{attribute 'linkalways'} 
{attribute 'no_explicit_call' := 'This FB is a CLASS and must be accessed using methods or properties'}
{attribute 'enable_dynamic_creation'}
FUNCTION_BLOCK Node_F_VN_WarpPerspective_Point EXTENDS VisionNode
VAR
	aSrcPoint : _TcVnPoint2_LREAL;
    aDestPoint : _TcVnPoint2_LREAL;
    aTransformationMatrix : _TcVnMatrix3x3_LREAL;
    hrPrev : _HRESULT(S_OK);
	hresult : _HRESULT(S_OK);
END_VAR

METHOD PUBLIC  Clone : I_Node
VAR
	pNode : POINTER TO Node_F_VN_WarpPerspective_Point;
END_VAR
pNode := __NEW(Node_F_VN_WarpPerspective_Point);
Clone := pNode^;
END_METHOD

METHOD FB_init : BOOL
VAR_INPUT
	bInitRetains : BOOL; // if TRUE, the retain variables are initialized (warm start / cold start)
	bInCopyCode : BOOL;  // if TRUE, the instance afterwards gets moved into the copy code (online change)
END_VAR
AddInput('aSrcPoint', aSrcPoint);
AddInput('aTransformationMatrix', aTransformationMatrix);
AddInput('hrPrev', hrPrev);
AddOutput('aDestPoint', aDestPoint);
AddOutput('hresult',hresult);
END_METHOD

METHOD PROTECTED OnExecute
hresult.Value := F_VN_WarpPerspective_Point(
	aSrcPoint := aSrcPoint.Value, 
	aDestPoint := aDestPoint.Value, 
	aTransformationMatrix := aTransformationMatrix.Value, 
	hrPrev := hrPrev.Value);
END_METHOD

METHOD PUBLIC PreExecutionCheck
VAR_INPUT
	Check : I_PreExecutionChecks;
END_VAR
END_METHOD

END_FUNCTION_BLOCK

(* stored: Version 1.1.0.1, ProductVersion 3.1.4024.13
   POU Node_F_VN_WarpPerspective_Point: Id {fe4a1952-b3e6-05fd-3595-0202b3859b2d}, SpecialFunc None
   Folder Constructor: Id {9918f522-b7af-0c35-2a84-ce1e1f478a3a}
   Method Clone: Id {32785e73-6b15-0187-0aae-8e91f868fbaf}
   Method FB_init: Id {12d9c296-436c-0ab1-2147-a13a0768f476}
   Method OnExecute: Id {eecfecbb-2588-0d41-2541-47045ce5101d}
   Method PreExecutionCheck: Id {90ad412e-b866-0692-2b3e-bbc0bfee69da} *)
